// Mitsubishi GX Works2 project: GX W2 L2 Ex 2 DK c   PLC: FX3G

// global labels: Global1
VAR_GLOBAL
  iBooster_SW AT X001 : BOOL;
  oExtraction_Fan AT Y001 : BOOL;
END_VAR

// task Task_01 (event TRUE, interval 0, priority 31): POU_01

PROGRAM POU_01
VAR
  TOF_1 : TOF;
END_VAR
(* structured ladder/FBD written out as ST: instructions are called as NAME(EN, inputs, outputs); _pN, _eN, _tN stand for wires *)
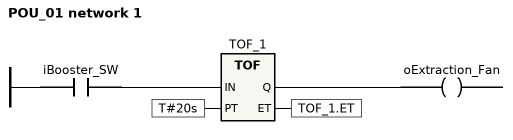
(* network 1 *)
TOF_1(IN := iBooster_SW, PT := T#20s, ET => TOF_1.ET);
oExtraction_Fan := TOF_1.Q;
END_PROGRAM
